(*
Searches an `I_Entity` for a `I_State` component matching provided id pattern.
Result:
- Ok - Returns `I_State`.
- None - Returns null.
- Err.Itf0 - Returns null, incorrect interface.
*)
FUNCTION GetState : Result
VAR_INPUT
	iEntity		: I_Entity;
	sTagId		: Str;
END_VAR
VAR_OUTPUT
	iState		: I_State;
END_VAR
VAR
	i			: Iter(1);
	_iComp		: I_FatComponent;
	cmp			: TagCmp;
END_VAR

IF iEntity = 0 THEN
	GetState := Err.Itf0;
	RETURN;
END_IF

WHILE IsOk(iEntity.Get(i.Next(), iComp => _iComp)) DO
	IF IsOk(ICompToIState(_iComp.Raw, iDest => iState)) THEN
		IF cmp.Set(iState.Tag).MatchWcdId(sTagId).IsTrue() THEN
			GetState := Ok;
			RETURN;
		ELSE
			iState := 0;
		END_IF
	END_IF
END_WHILE

END_FUNCTION

(* stored: Version 1.1.0.1
   POU GetState: Id {4a6ca9b6-95b3-4d02-9450-013f1847a076}, SpecialFunc None *)
